// TIA Portal project "Robocik" (V16)
// Robot Mitsubishi

(* hardware
DEVICE "S7-1200 station_1"  S7-1200 Station
   slot 0: "Rack_0"  S7-1200 Rack  Rack  V1.0
   slot 1: "CRnD-7xx/CR75x-D"  CPU 1212C AC/DC/Rly  6ES7 212-1BE40-0XB0  V4.3
   slot 2: "DI 16/DQ 16x24VDC_1"  6ES7 223-1BL32-0XB0  V2.0
DEVICE "HMI_1"  TP1500 Comfort
   slot 0: "HMI_1"  TP1500 Comfort  6AV2 124-0QC02-0AX0  16.0.0.0
   slot 1: "HMI_RT_1"  TP1500 Comfort  6AV2 124-0QC02-0AX0  16.0.0.0
   slot 5: "HMI_1.IE_CP_1"  PROFINET Interface  16.0.0.0
      slot 1: "PROFINET Interface_1"  PROFINET Interface
         slot 1: "Port_1"  Port
         slot 2: "Port_2"  Port
   slot 6: "HMI_1.IE_CP_2"  PROFINET Interface  16.0.0.0
      slot 1: "PROFINET Interface_GBit"  PROFINET Interface
         slot 1: "Port_1"  Port
   slot 7: "HMI_1.MPI/DP_CP_1"  MPI/DP Interface  16.0.0.0
*)

// ===== PLC "CRnD-7xx/CR75x-D"  CPU 1212C AC/DC/Rly =====

VAR_GLOBAL   // PLC tag table "Default tag table"
   "Sensor 1" AT %I9.0 : Bool;
   "Sensor 2" AT %I9.1 : Bool;
   "Sensor 3" AT %I9.2 : Bool;
   "Sensor 4" AT %I9.3 : Bool;
   "Sensor 5" AT %I9.4 : Bool;
   "StackLight_GreenLight" AT %Q9.0 : Bool;
   "StackLight_RedLight" AT %Q9.1 : Bool;
   "Actuator_1_Set" AT %Q0.0 : Bool;
   "Actuator_1_Reset" AT %Q0.1 : Bool;
   "Actuator_2_Set" AT %Q0.2 : Bool;
   "Actuator_2_Reset" AT %Q0.3 : Bool;
   "Actuator_3_Set" AT %Q0.4 : Bool;
   "Actuator_3_Reset" AT %Q0.5 : Bool;
   "Actuator_1_HomePosition" AT %I0.0 : Bool;
   "Actuator_2_HomePosition" AT %I0.2 : Bool;
   "Actuator_3_HomePosition" AT %I0.4 : Bool;
   "Actuator_1_WorkPosition" AT %I0.1 : Bool;
   "Actuator_2_WorkPosition" AT %I0.3 : Bool;
   "Actuator_3_WorkPosition" AT %I0.5 : Bool;
   "Robot_Input_8" AT %Q8.0 : Bool;
   "Robot_Input_9" AT %Q8.1 : Bool;
   "Robot_Input_10" AT %Q8.2 : Bool;
   "Robot_Input_11" AT %Q8.3 : Bool;
   "Robot_Input_12" AT %Q8.4 : Bool;
   "Robot_Input_13" AT %Q8.5 : Bool;
   "Robot_Input_14" AT %Q8.6 : Bool;
   "Robot_Input_15" AT %Q8.7 : Bool;
   "Robot_Output_8" AT %I8.0 : Bool;
   "Robot_Output_9" AT %I8.1 : Bool;
   "Robot_Output_10" AT %I8.2 : Bool;
   "Robot_Output_11" AT %I8.3 : Bool;
   "Robot_Output_12" AT %I8.4 : Bool;
   "Robot_Output_13" AT %I8.5 : Bool;
   "Robot_Output_14" AT %I8.6 : Bool;
   "Robot_Output_15" AT %I8.7 : Bool;
   "Robot_Output_2_Fault" AT %I0.6 : Bool;
   "Sensor 6" AT %I9.5 : Bool;
END_VAR

DATA_BLOCK "DB_HMICommands"   // DB1
{ S7_Optimized_Access := 'TRUE' }
VERSION : 0.1
   VAR
      ControPanel : Struct
         Start : Bool;
         Stop : Bool;
         Reset : Bool;
      END_STRUCT;
   END_VAR
BEGIN
END_DATA_BLOCK

DATA_BLOCK "DB_Configuration"   // DB2
{ S7_Optimized_Access := 'TRUE' }
VERSION : 0.1
   VAR
      Actuator_1 : Struct
         InterlockForward : Bool;
         InterlockBAckword : Bool;
      END_STRUCT;
      Actuator_2 : Struct
         InterlockForward : Bool;
         InterlockBAckword : Bool;
      END_STRUCT;
      Actuator_3 : Struct
         InterlockForward : Bool;
         InterlockBAckword : Bool;
      END_STRUCT;
   END_VAR
BEGIN
END_DATA_BLOCK

DATA_BLOCK "DB_Actuator_1"   // DB3
{ S7_Optimized_Access := 'TRUE' }
VERSION : 0.1
// stored: InstanceOfName FB_Actuator
"FB_Actuator"
BEGIN
END_DATA_BLOCK

DATA_BLOCK "DB_Actuator_2"   // DB4
{ S7_Optimized_Access := 'TRUE' }
VERSION : 0.1
// stored: InstanceOfName FB_Actuator
"FB_Actuator"
BEGIN
END_DATA_BLOCK

DATA_BLOCK "DB_Actuator_3"   // DB5
{ S7_Optimized_Access := 'TRUE' }
VERSION : 0.1
// stored: InstanceOfName FB_Actuator
"FB_Actuator"
BEGIN
END_DATA_BLOCK

DATA_BLOCK "FB_First_Actuator_DB"   // DB7
{ S7_Optimized_Access := 'TRUE' }
VERSION : 0.1
// stored: InstanceOfName FB_First_Actuator
"FB_First_Actuator"
BEGIN
END_DATA_BLOCK

DATA_BLOCK "FB_Rotation_DB"   // DB9
{ S7_Optimized_Access := 'TRUE' }
VERSION : 0.1
// stored: InstanceOfName FB_Rotation
"FB_Rotation"
BEGIN
END_DATA_BLOCK

DATA_BLOCK "FB_Cheack_For_Hole_DB"   // DB10
{ S7_Optimized_Access := 'TRUE' }
VERSION : 0.1
// stored: InstanceOfName FB_Cheack_For_Hole
"FB_Cheack_For_Hole"
BEGIN
END_DATA_BLOCK

DATA_BLOCK "FB_Metal_Detector_DB"   // DB11
{ S7_Optimized_Access := 'TRUE' }
VERSION : 0.1
// stored: InstanceOfName FB_Metal_Detector
"FB_Metal_Detector"
BEGIN
END_DATA_BLOCK

DATA_BLOCK "FB_Resting_For_Disc_DB"   // DB12
{ S7_Optimized_Access := 'TRUE' }
VERSION : 0.1
// stored: InstanceOfName FB_Resting_For_Disc
"FB_Resting_For_Disc"
BEGIN
END_DATA_BLOCK

DATA_BLOCK "FB_HMI_Control_DB"   // DB13
{ S7_Optimized_Access := 'TRUE' }
VERSION : 0.1
// stored: InstanceOfName FB_HMI_Control
"FB_HMI_Control"
BEGIN
END_DATA_BLOCK

DATA_BLOCK "DB_Work"   // DB14
{ S7_Optimized_Access := 'TRUE' }
VERSION : 0.1
   VAR
      Actu1 : Struct
         InterlockForward : Bool;
         InterlockBAckward : Bool;
      END_STRUCT;
      Actu2 : Struct
         InterlockForward : Bool;
         InterlockBAckward : Bool;
      END_STRUCT;
      Actu3 : Struct
         InterlockForward : Bool;
         InterlockBAckward : Bool;
      END_STRUCT;
   END_VAR
BEGIN
END_DATA_BLOCK

FUNCTION_BLOCK "FB_Actuator"   // FB1, LAD
{ S7_Optimized_Access := 'TRUE' }
VERSION : 0.1
   VAR_INPUT
      ix_InterlockForward : Bool;
      ix_InterlockBackword : Bool;
   END_VAR
   VAR_OUTPUT
      iqx_MoveFarword : Bool;
      iqx_MoveBackword : Bool;
   END_VAR
BEGIN

REGION Network 1
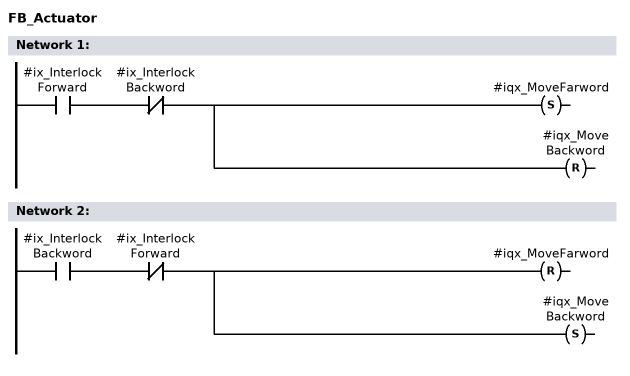
   RUNG wire#powerrail
      Contact( #ix_InterlockForward )
      I_Contact( #ix_InterlockBackword )
      wire#w1
      S_Coil( #iqx_MoveFarword )
   END_RUNG
   RUNG wire#w1
      R_Coil( #iqx_MoveBackword )
   END_RUNG
   // the same network as SCL:
   IF #ix_InterlockForward AND NOT #ix_InterlockBackword THEN
       #iqx_MoveFarword := TRUE;
       #iqx_MoveBackword := FALSE;
   END_IF;
END_REGION

REGION Network 2
   RUNG wire#powerrail
      Contact( #ix_InterlockBackword )
      I_Contact( #ix_InterlockForward )
      wire#w1
      R_Coil( #iqx_MoveFarword )
   END_RUNG
   RUNG wire#w1
      S_Coil( #iqx_MoveBackword )
   END_RUNG
   // the same network as SCL:
   IF #ix_InterlockBackword AND NOT #ix_InterlockForward THEN
       #iqx_MoveFarword := FALSE;
       #iqx_MoveBackword := TRUE;
   END_IF;
END_REGION
END_FUNCTION_BLOCK

FUNCTION_BLOCK "FB_HMI_Control"   // FB2, LAD
{ S7_Optimized_Access := 'TRUE' }
VERSION : 0.1
   VAR_INPUT
      ix_StartFeedback : Bool;
      ix_StopFeedback : Bool;
   END_VAR
   VAR_IN_OUT
      iqx_StartRobot : Bool;
      iqx_StopRobot : Bool;
   END_VAR
BEGIN

REGION Network 1
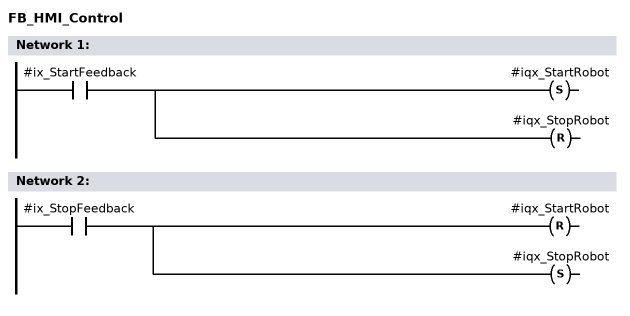
   RUNG wire#powerrail
      Contact( #ix_StartFeedback )
      wire#w1
      S_Coil( #iqx_StartRobot )
   END_RUNG
   RUNG wire#w1
      R_Coil( #iqx_StopRobot )
   END_RUNG
   // the same network as SCL:
   IF #ix_StartFeedback THEN
       #iqx_StartRobot := TRUE;
       #iqx_StopRobot := FALSE;
   END_IF;
END_REGION

REGION Network 2
   RUNG wire#powerrail
      Contact( #ix_StopFeedback )
      wire#w1
      R_Coil( #iqx_StartRobot )
   END_RUNG
   RUNG wire#w1
      S_Coil( #iqx_StopRobot )
   END_RUNG
   // the same network as SCL:
   IF #ix_StopFeedback THEN
       #iqx_StartRobot := FALSE;
       #iqx_StopRobot := TRUE;
   END_IF;
END_REGION
END_FUNCTION_BLOCK

FUNCTION_BLOCK "FB_Metal_Detector"   // FB3, LAD
{ S7_Optimized_Access := 'TRUE' }
VERSION : 0.1
   VAR_INPUT
      ix_CheackPosition : Bool;
      ix_MetalSensor : Bool;
   END_VAR
   VAR_OUTPUT
      qx_RobotInput12 : Bool;
   END_VAR
BEGIN

REGION Network 1
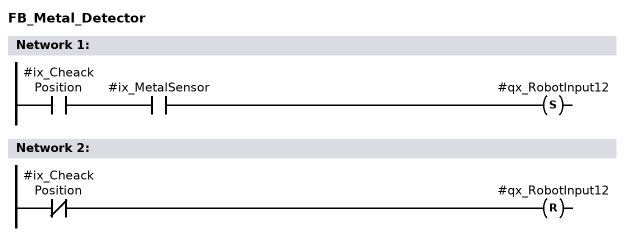
   RUNG wire#powerrail
      Contact( #ix_CheackPosition )
      Contact( #ix_MetalSensor )
      S_Coil( #qx_RobotInput12 )
   END_RUNG
   // the same network as SCL:
   IF #ix_CheackPosition AND #ix_MetalSensor THEN #qx_RobotInput12 := TRUE; END_IF;
END_REGION

REGION Network 2
   RUNG wire#powerrail
      I_Contact( #ix_CheackPosition )
      R_Coil( #qx_RobotInput12 )
   END_RUNG
   // the same network as SCL:
   IF NOT #ix_CheackPosition THEN #qx_RobotInput12 := FALSE; END_IF;
END_REGION
END_FUNCTION_BLOCK

FUNCTION_BLOCK "FB_Cheack_For_Hole"   // FB4, LAD
{ S7_Optimized_Access := 'TRUE' }
VERSION : 0.1
   VAR_INPUT
      ix_CheackPosition : Bool;
      ix_LAser : Bool;
   END_VAR
   VAR_OUTPUT
      qx_RobotInput11 : Bool;
   END_VAR
BEGIN

REGION Network 1
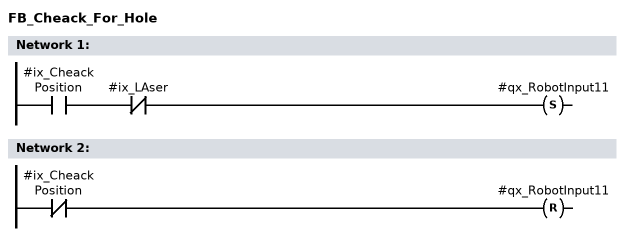
   RUNG wire#powerrail
      Contact( #ix_CheackPosition )
      I_Contact( #ix_LAser )
      S_Coil( #qx_RobotInput11 )
   END_RUNG
   // the same network as SCL:
   IF #ix_CheackPosition AND NOT #ix_LAser THEN #qx_RobotInput11 := TRUE; END_IF;
END_REGION

REGION Network 2
   RUNG wire#powerrail
      I_Contact( #ix_CheackPosition )
      R_Coil( #qx_RobotInput11 )
   END_RUNG
   // the same network as SCL:
   IF NOT #ix_CheackPosition THEN #qx_RobotInput11 := FALSE; END_IF;
END_REGION
END_FUNCTION_BLOCK

FUNCTION_BLOCK "FB_Resting_For_Disc"   // FB5, LAD
{ S7_Optimized_Access := 'TRUE' }
VERSION : 0.1
   VAR_INPUT
      ix_RobotOutput12 : Bool;
      ix_B5 : Bool;
      ix_B6 : Bool;
      ix_StartRobot : Bool;
   END_VAR
   VAR_OUTPUT
      ix_RobotInput13 : Bool;
   END_VAR
   VAR_IN_OUT
      iqx_InterlockForward : Bool;
      iqx_InterlockBackward : Bool;
   END_VAR
BEGIN

REGION Network 1
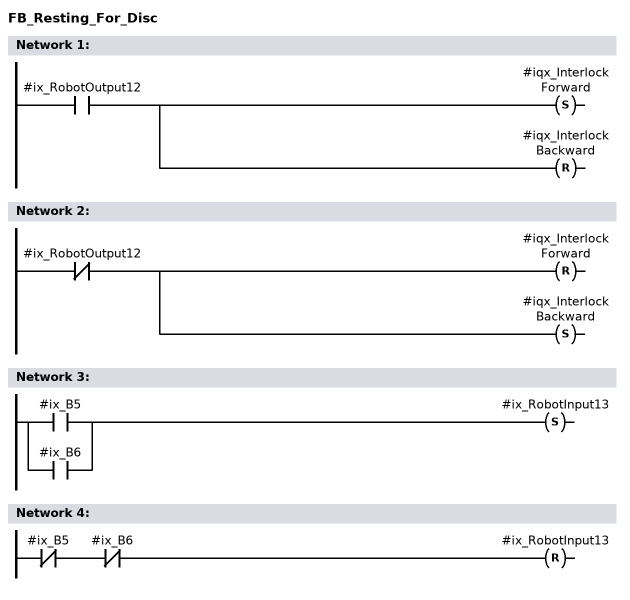
   RUNG wire#powerrail
      Contact( #ix_RobotOutput12 )
      wire#w1
      S_Coil( #iqx_InterlockForward )
   END_RUNG
   RUNG wire#w1
      R_Coil( #iqx_InterlockBackward )
   END_RUNG
   // the same network as SCL:
   IF #ix_RobotOutput12 THEN
       #iqx_InterlockForward := TRUE;
       #iqx_InterlockBackward := FALSE;
   END_IF;
END_REGION

REGION Network 2
   RUNG wire#powerrail
      I_Contact( #ix_RobotOutput12 )
      wire#w1
      R_Coil( #iqx_InterlockForward )
   END_RUNG
   RUNG wire#w1
      S_Coil( #iqx_InterlockBackward )
   END_RUNG
   // the same network as SCL:
   IF NOT #ix_RobotOutput12 THEN
       #iqx_InterlockForward := FALSE;
       #iqx_InterlockBackward := TRUE;
   END_IF;
END_REGION

REGION Network 3
   RUNG wire#powerrail
      Contact( #ix_B5 )
      wire#w1
      S_Coil( #ix_RobotInput13 )
   END_RUNG
   RUNG wire#powerrail
      Contact( #ix_B6 )
   END_RUNG wire#w1
   // the same network as SCL:
   IF #ix_B5 OR #ix_B6 THEN #ix_RobotInput13 := TRUE; END_IF;
END_REGION

REGION Network 4
   RUNG wire#powerrail
      I_Contact( #ix_B5 )
      I_Contact( #ix_B6 )
      R_Coil( #ix_RobotInput13 )
   END_RUNG
   // the same network as SCL:
   IF NOT #ix_B5 AND NOT #ix_B6 THEN #ix_RobotInput13 := FALSE; END_IF;
END_REGION
END_FUNCTION_BLOCK

FUNCTION_BLOCK "FB_Rotation"   // FB6, LAD
{ S7_Optimized_Access := 'TRUE' }
VERSION : 0.1
   VAR_INPUT
      ix_RobotOutput8 : Bool;
      ix_RobotOutput9 : Bool;
      ix_Actuator_2_HomePosition : Bool;
      ix_Actuator_2_WorkPosition : Bool;
      ix_B5 : Bool;
      ix_B6 : Bool;
      ix_RobotOutput12 : Bool;
   END_VAR
   VAR_OUTPUT
      qx_RobotInput10 : Bool;
   END_VAR
   VAR_IN_OUT
      iqx_InterlockForward : Bool;
      iqx_InterlockBackward : Bool;
   END_VAR
   VAR
      s_TON_Timer : TON_TIME;
      s_TON_Timer_1 : TON_TIME;
   END_VAR
BEGIN

REGION Network 1
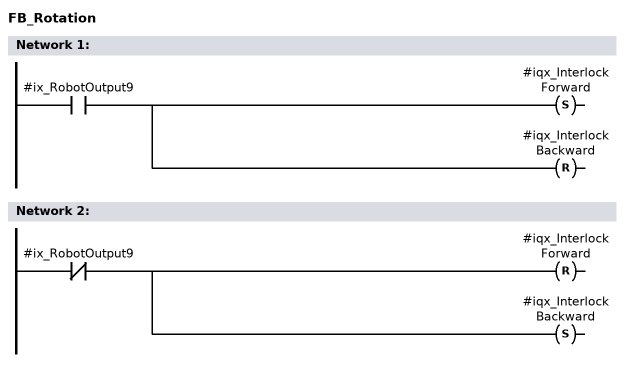
   RUNG wire#powerrail
      Contact( #ix_RobotOutput9 )
      wire#w1
      S_Coil( #iqx_InterlockForward )
   END_RUNG
   RUNG wire#w1
      R_Coil( #iqx_InterlockBackward )
   END_RUNG
   // the same network as SCL:
   IF #ix_RobotOutput9 THEN
       #iqx_InterlockForward := TRUE;
       #iqx_InterlockBackward := FALSE;
   END_IF;
END_REGION

REGION Network 2
   RUNG wire#powerrail
      I_Contact( #ix_RobotOutput9 )
      wire#w1
      R_Coil( #iqx_InterlockForward )
   END_RUNG
   RUNG wire#w1
      S_Coil( #iqx_InterlockBackward )
   END_RUNG
   // the same network as SCL:
   IF NOT #ix_RobotOutput9 THEN
       #iqx_InterlockForward := FALSE;
       #iqx_InterlockBackward := TRUE;
   END_IF;
END_REGION
END_FUNCTION_BLOCK

FUNCTION_BLOCK "FB_First_Actuator"   // FB7, LAD
{ S7_Optimized_Access := 'TRUE' }
VERSION : 0.1
   VAR_INPUT
      ix_B1 : Bool;
      ix_B2 : Bool;
      ix_Act_1_HomePosition : Bool;
      ix_Act_1_WorkPosition : Bool;
      ix_RobotOutput15 : Bool;
      ix_StartRobot : Bool;
      ix_RobotOutput14 : Bool;
   END_VAR
   VAR_OUTPUT
      qx_Output_8_Robot : Bool;
      qx_Output_9_Robot : Bool;
      ix_Output_15_Robot : Bool;
   END_VAR
   VAR_IN_OUT
      iqx_StartStop : Bool;
      iqx_InterlockForward : Bool;
      iqx_InterlockBackword : Bool;
   END_VAR
   VAR
      sx_Start : Bool;
      sx_ptrig : Bool;
   END_VAR
BEGIN

REGION Network 1: Start ( info from robot)
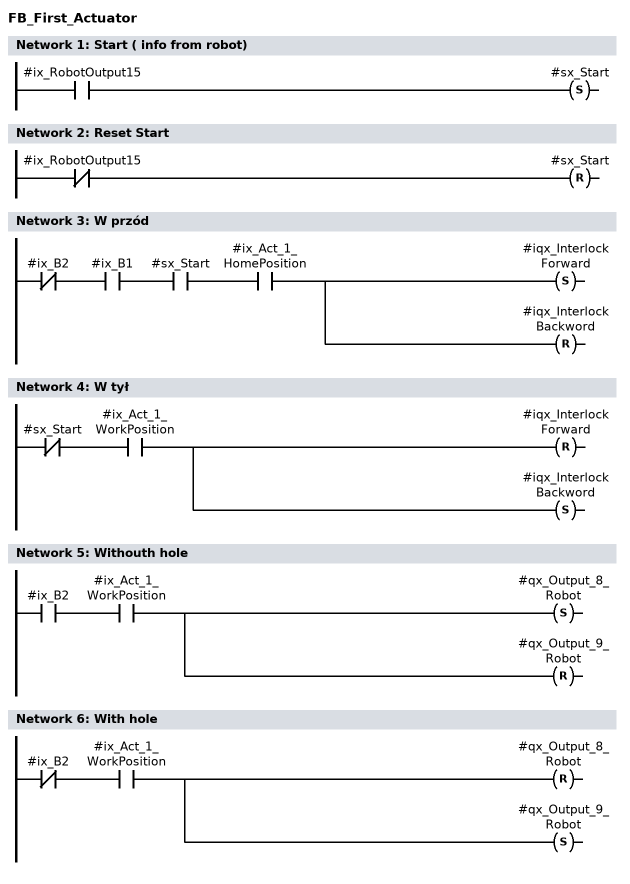
   RUNG wire#powerrail
      Contact( #ix_RobotOutput15 )
      S_Coil( #sx_Start )
   END_RUNG
   // the same network as SCL:
   IF #ix_RobotOutput15 THEN #sx_Start := TRUE; END_IF;
END_REGION

REGION Network 2: Reset Start
   RUNG wire#powerrail
      I_Contact( #ix_RobotOutput15 )
      R_Coil( #sx_Start )
   END_RUNG
   // the same network as SCL:
   IF NOT #ix_RobotOutput15 THEN #sx_Start := FALSE; END_IF;
END_REGION

REGION Network 3: W przód
   RUNG wire#powerrail
      I_Contact( #ix_B2 )
      Contact( #ix_B1 )
      Contact( #sx_Start )
      Contact( #ix_Act_1_HomePosition )
      wire#w1
      S_Coil( #iqx_InterlockForward )
   END_RUNG
   RUNG wire#w1
      R_Coil( #iqx_InterlockBackword )
   END_RUNG
   // the same network as SCL:
   IF NOT #ix_B2 AND #ix_B1 AND #sx_Start AND #ix_Act_1_HomePosition THEN
       #iqx_InterlockForward := TRUE;
       #iqx_InterlockBackword := FALSE;
   END_IF;
END_REGION

REGION Network 4: W tył
   RUNG wire#powerrail
      I_Contact( #sx_Start )
      Contact( #ix_Act_1_WorkPosition )
      wire#w1
      R_Coil( #iqx_InterlockForward )
   END_RUNG
   RUNG wire#w1
      S_Coil( #iqx_InterlockBackword )
   END_RUNG
   // the same network as SCL:
   IF NOT #sx_Start AND #ix_Act_1_WorkPosition THEN
       #iqx_InterlockForward := FALSE;
       #iqx_InterlockBackword := TRUE;
   END_IF;
END_REGION

REGION Network 5: Withouth hole
   RUNG wire#powerrail
      Contact( #ix_B2 )
      Contact( #ix_Act_1_WorkPosition )
      wire#w1
      S_Coil( #qx_Output_8_Robot )
   END_RUNG
   RUNG wire#w1
      R_Coil( #qx_Output_9_Robot )
   END_RUNG
   // the same network as SCL:
   IF #ix_B2 AND #ix_Act_1_WorkPosition THEN
       #qx_Output_8_Robot := TRUE;
       #qx_Output_9_Robot := FALSE;
   END_IF;
END_REGION

REGION Network 6: With hole
   RUNG wire#powerrail
      I_Contact( #ix_B2 )
      Contact( #ix_Act_1_WorkPosition )
      wire#w1
      R_Coil( #qx_Output_8_Robot )
   END_RUNG
   RUNG wire#w1
      S_Coil( #qx_Output_9_Robot )
   END_RUNG
   // the same network as SCL:
   IF NOT #ix_B2 AND #ix_Act_1_WorkPosition THEN
       #qx_Output_8_Robot := FALSE;
       #qx_Output_9_Robot := TRUE;
   END_IF;
END_REGION
END_FUNCTION_BLOCK

FUNCTION "FC_Area" : Void   // FC1, LAD
{ S7_Optimized_Access := 'TRUE' }
VERSION : 0.1
BEGIN

REGION Network 1: HMI
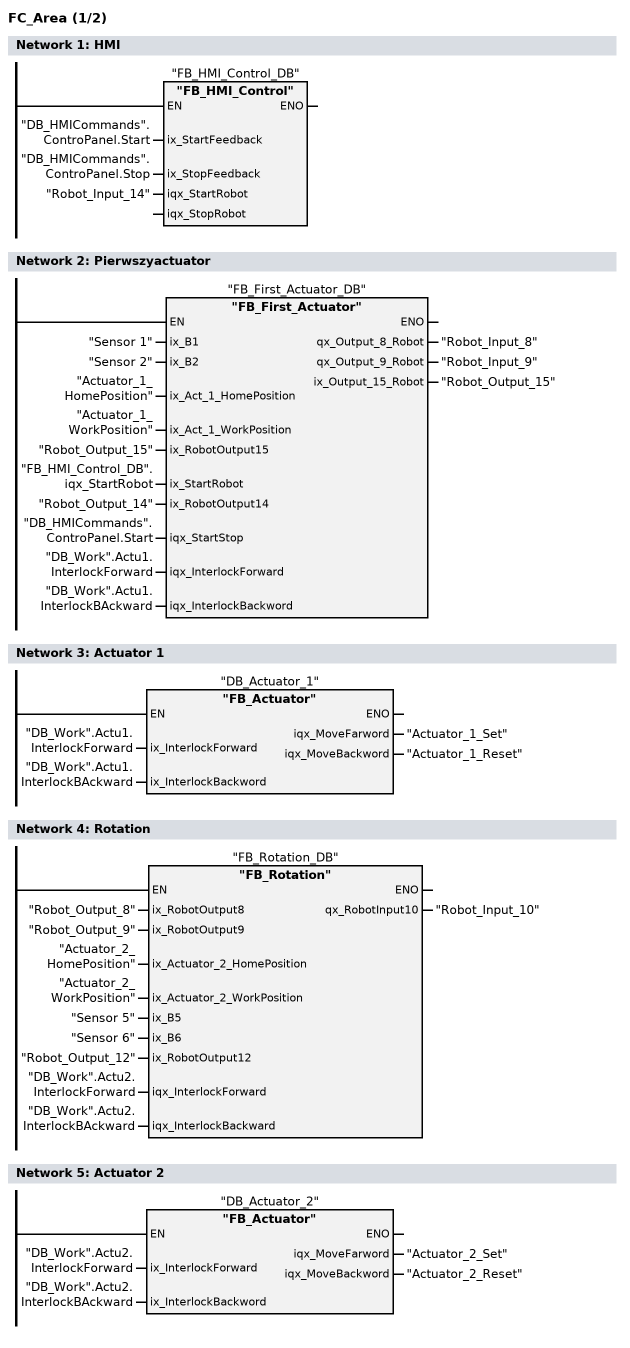
   RUNG wire#powerrail
      "FB_HMI_Control_DB"(ix_StartFeedback := "DB_HMICommands".ControPanel.Start, ix_StopFeedback := "DB_HMICommands".ControPanel.Stop, iqx_StartRobot := "Robot_Input_14", iqx_StopRobot :=)
   END_RUNG
   // the same network as SCL:
   "FB_HMI_Control_DB"(ix_StartFeedback := "DB_HMICommands".ControPanel.Start,   // "FB_HMI_Control"
                       ix_StopFeedback := "DB_HMICommands".ControPanel.Stop,
                       iqx_StartRobot := "Robot_Input_14");
END_REGION

REGION Network 2: Pierwszyactuator
   RUNG wire#powerrail
      "FB_First_Actuator_DB"(ix_B1 := "Sensor 1", ix_B2 := "Sensor 2", ix_Act_1_HomePosition := "Actuator_1_HomePosition", ix_Act_1_WorkPosition := "Actuator_1_WorkPosition", ix_RobotOutput15 := "Robot_Output_15", ix_StartRobot := "FB_HMI_Control_DB".iqx_StartRobot, ix_RobotOutput14 := "Robot_Output_14", iqx_StartStop := "DB_HMICommands".ControPanel.Start, iqx_InterlockForward := "DB_Work".Actu1.InterlockForward, iqx_InterlockBackword := "DB_Work".Actu1.InterlockBAckward, qx_Output_8_Robot => "Robot_Input_8", qx_Output_9_Robot => "Robot_Input_9", ix_Output_15_Robot => "Robot_Output_15")
   END_RUNG
   // the same network as SCL:
   "FB_First_Actuator_DB"(ix_B1 := "Sensor 1",   // "FB_First_Actuator"
                          ix_B2 := "Sensor 2",
                          ix_Act_1_HomePosition := "Actuator_1_HomePosition",
                          ix_Act_1_WorkPosition := "Actuator_1_WorkPosition",
                          ix_RobotOutput15 := "Robot_Output_15",
                          ix_StartRobot := "FB_HMI_Control_DB".iqx_StartRobot,
                          ix_RobotOutput14 := "Robot_Output_14",
                          iqx_StartStop := "DB_HMICommands".ControPanel.Start,
                          iqx_InterlockForward := "DB_Work".Actu1.InterlockForward,
                          iqx_InterlockBackword := "DB_Work".Actu1.InterlockBAckward,
                          qx_Output_8_Robot => "Robot_Input_8",
                          qx_Output_9_Robot => "Robot_Input_9",
                          ix_Output_15_Robot => "Robot_Output_15");
END_REGION

REGION Network 3: Actuator 1
   RUNG wire#powerrail
      "DB_Actuator_1"(ix_InterlockForward := "DB_Work".Actu1.InterlockForward, ix_InterlockBackword := "DB_Work".Actu1.InterlockBAckward, iqx_MoveFarword => "Actuator_1_Set", iqx_MoveBackword => "Actuator_1_Reset")
   END_RUNG
   // the same network as SCL:
   "DB_Actuator_1"(ix_InterlockForward := "DB_Work".Actu1.InterlockForward,   // "FB_Actuator"
                   ix_InterlockBackword := "DB_Work".Actu1.InterlockBAckward,
                   iqx_MoveFarword => "Actuator_1_Set",
                   iqx_MoveBackword => "Actuator_1_Reset");
END_REGION

REGION Network 4: Rotation
   RUNG wire#powerrail
      "FB_Rotation_DB"(ix_RobotOutput8 := "Robot_Output_8", ix_RobotOutput9 := "Robot_Output_9", ix_Actuator_2_HomePosition := "Actuator_2_HomePosition", ix_Actuator_2_WorkPosition := "Actuator_2_WorkPosition", ix_B5 := "Sensor 5", ix_B6 := "Sensor 6", ix_RobotOutput12 := "Robot_Output_12", iqx_InterlockForward := "DB_Work".Actu2.InterlockForward, iqx_InterlockBackward := "DB_Work".Actu2.InterlockBAckward, qx_RobotInput10 => "Robot_Input_10")
   END_RUNG
   // the same network as SCL:
   "FB_Rotation_DB"(ix_RobotOutput8 := "Robot_Output_8",   // "FB_Rotation"
                    ix_RobotOutput9 := "Robot_Output_9",
                    ix_Actuator_2_HomePosition := "Actuator_2_HomePosition",
                    ix_Actuator_2_WorkPosition := "Actuator_2_WorkPosition",
                    ix_B5 := "Sensor 5",
                    ix_B6 := "Sensor 6",
                    ix_RobotOutput12 := "Robot_Output_12",
                    iqx_InterlockForward := "DB_Work".Actu2.InterlockForward,
                    iqx_InterlockBackward := "DB_Work".Actu2.InterlockBAckward,
                    qx_RobotInput10 => "Robot_Input_10");
END_REGION

REGION Network 5: Actuator 2
   RUNG wire#powerrail
      "DB_Actuator_2"(ix_InterlockForward := "DB_Work".Actu2.InterlockForward, ix_InterlockBackword := "DB_Work".Actu2.InterlockBAckward, iqx_MoveFarword => "Actuator_2_Set", iqx_MoveBackword => "Actuator_2_Reset")
   END_RUNG
   // the same network as SCL:
   "DB_Actuator_2"(ix_InterlockForward := "DB_Work".Actu2.InterlockForward,   // "FB_Actuator"
                   ix_InterlockBackword := "DB_Work".Actu2.InterlockBAckward,
                   iqx_MoveFarword => "Actuator_2_Set",
                   iqx_MoveBackword => "Actuator_2_Reset");
END_REGION

REGION Network 6: Cheack for holes
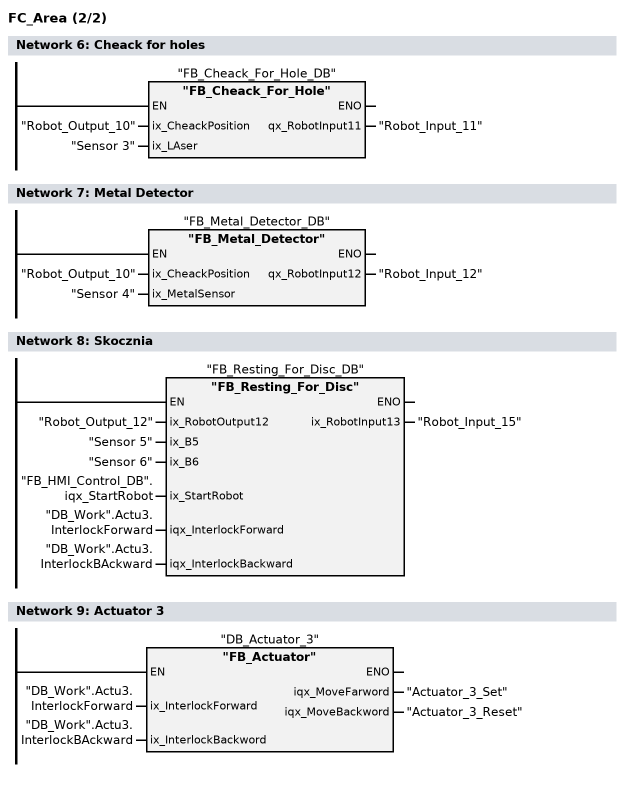
   RUNG wire#powerrail
      "FB_Cheack_For_Hole_DB"(ix_CheackPosition := "Robot_Output_10", ix_LAser := "Sensor 3", qx_RobotInput11 => "Robot_Input_11")
   END_RUNG
   // the same network as SCL:
   "FB_Cheack_For_Hole_DB"(ix_CheackPosition := "Robot_Output_10",   // "FB_Cheack_For_Hole"
                           ix_LAser := "Sensor 3",
                           qx_RobotInput11 => "Robot_Input_11");
END_REGION

REGION Network 7: Metal Detector
   RUNG wire#powerrail
      "FB_Metal_Detector_DB"(ix_CheackPosition := "Robot_Output_10", ix_MetalSensor := "Sensor 4", qx_RobotInput12 => "Robot_Input_12")
   END_RUNG
   // the same network as SCL:
   "FB_Metal_Detector_DB"(ix_CheackPosition := "Robot_Output_10",   // "FB_Metal_Detector"
                          ix_MetalSensor := "Sensor 4",
                          qx_RobotInput12 => "Robot_Input_12");
END_REGION

REGION Network 8: Skocznia
   RUNG wire#powerrail
      "FB_Resting_For_Disc_DB"(ix_RobotOutput12 := "Robot_Output_12", ix_B5 := "Sensor 5", ix_B6 := "Sensor 6", ix_StartRobot := "FB_HMI_Control_DB".iqx_StartRobot, iqx_InterlockForward := "DB_Work".Actu3.InterlockForward, iqx_InterlockBackward := "DB_Work".Actu3.InterlockBAckward, ix_RobotInput13 => "Robot_Input_15")
   END_RUNG
   // the same network as SCL:
   "FB_Resting_For_Disc_DB"(ix_RobotOutput12 := "Robot_Output_12",   // "FB_Resting_For_Disc"
                           ix_B5 := "Sensor 5",
                           ix_B6 := "Sensor 6",
                           ix_StartRobot := "FB_HMI_Control_DB".iqx_StartRobot,
                           iqx_InterlockForward := "DB_Work".Actu3.InterlockForward,
                           iqx_InterlockBackward := "DB_Work".Actu3.InterlockBAckward,
                           ix_RobotInput13 => "Robot_Input_15");
END_REGION

REGION Network 9: Actuator 3
   RUNG wire#powerrail
      "DB_Actuator_3"(ix_InterlockForward := "DB_Work".Actu3.InterlockForward, ix_InterlockBackword := "DB_Work".Actu3.InterlockBAckward, iqx_MoveFarword => "Actuator_3_Set", iqx_MoveBackword => "Actuator_3_Reset")
   END_RUNG
   // the same network as SCL:
   "DB_Actuator_3"(ix_InterlockForward := "DB_Work".Actu3.InterlockForward,   // "FB_Actuator"
                   ix_InterlockBackword := "DB_Work".Actu3.InterlockBAckward,
                   iqx_MoveFarword => "Actuator_3_Set",
                   iqx_MoveBackword => "Actuator_3_Reset");
END_REGION
END_FUNCTION

ORGANIZATION_BLOCK "Main"   // OB1, LAD, ProgramCycle
TITLE = "Main Program Sweep (Cycle)"
{ S7_Optimized_Access := 'TRUE' }
VERSION : 0.1
BEGIN

REGION Network 1
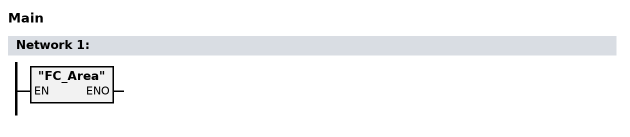
   RUNG wire#powerrail
      "FC_Area"()
   END_RUNG
   // the same network as SCL:
   "FC_Area"();
END_REGION
END_ORGANIZATION_BLOCK

(* ===== HMI "HMI_RT_1" =====
system functions are stored by id; their names below are inferred from use
connection "HMI_Connection_1": ETHERNET, S7_1200_OMS

Template "Template_1" 1280x800
   Button "Exit" at 1200,739 size 78x59; TextOff 'Exit'; PictureOff "ExitRuntime_TP1500_Comfort_TR"; PictureOn "ExitRuntime_TP1500_Comfort_TR"
      on Release: StopRuntime(0)
   Button "Template_Button" at 1120,739 size 78x59; TextOff 'Text'
   Button "Template_Button_1" at 1040,739 size 78x59; TextOff 'Text'
   Button "Template_Button_2" at 960,739 size 78x59; TextOff 'Text'
   Button "Template_Button_3" at 880,739 size 78x59; TextOff 'Text'
   Button "Template_Button_4" at 800,739 size 78x59; TextOff 'Text'
   Button "Template_Button_5" at 720,739 size 78x59; TextOff 'Text'
   Button "Template_Button_6" at 640,739 size 78x59; TextOff 'Text'
   Button "Template_Button_7" at 561,739 size 78x59; TextOff 'Text'
   Button "Template_Button_8" at 481,739 size 78x59; TextOff 'Text'
   Button "Template_Button_9" at 401,739 size 78x59; TextOff 'Text'
   Button "Template_Button_10" at 321,739 size 78x59; TextOff 'Text'
   Button "Template_Button_11" at 241,739 size 78x59; TextOff 'Text'
   Button "Template_Button_12" at 161,739 size 78x59; TextOff 'Text'
   Button "Template_Button_13" at 81,739 size 78x59; TextOff 'Factory'
      on Release: ActivateScreen("Factory", 0)
   Button "Start screen" at 1,739 size 78x59; TextOff 'Start screen'; PictureOff "NavigateHome_TP1500_Comfort_TR"; PictureOn "NavigateHome_TP1500_Comfort_TR"
      on Release: ActivateScreen("Main", 0)

screen "Main" 1280x800, template "Template_1"
   TextField "HmiScreenItemData" at 128,354 size 1024x27; Text 'Welcome to HMI_1 (TP1500 Comfort)!'

screen "Factory" 1280x800, template "Template_1"
   Button "Button_1" at 39,53 size 96x32; TextOff 'Start'
   Button "Button_2" at 39,99 size 96x32; TextOff 'Stop'
   Button "Button_3" at 40,143 size 96x32; TextOff 'Reset'
*)